// TIA Portal V21 export
TYPE "LAxisCtrl_typeOffset"
TITLE = LAxisCtrl_typeOffset
// Support: tech.team.motioncontrol@siemens.com
   STRUCT
      offset : LReal := 0.0;   // Absolute or relative offset shift
      profileReference : DInt := 1;   // Type of traversing of the following value offset (1: Traverse following value offset using leading value distance starting from the current effective leading value position; 2: Traverse following value offset using leading value distance from the effective leading value position "StartPosition"; 5: Cancel only one waiting job for the following value offset)
      offsetDistance : LReal;   // Effective leading value distance while traversing the following value offset when "ProfileReference" = 1, 2
      startPosition : LReal;   // Effective leading value position starting from which the following value offset is traversed when "ProfileReference" = 2
      direction : DInt := 3;   // Direction of the leading value distance (1: Positive direction; 2: Negative direction; 3: Current direction) when "ProfileReference" = 1, 2
      offsetAbsolute : Bool := TRUE;   // Indicates the type of the offset shift. TRUE: Shift the following value as an absolute shift; FALSE: Shift the following value relative to the existing following value shift
      offsetChangeOnTheFly : Bool := FALSE;   // TRUE: Changing offset shift on-the-fly at absolute offset shift. FALSE: Offset shift change requires a new rising edge at offset input
   END_STRUCT;
END_TYPE
